Yaskawa INFORM job: R1_W72(-45,-90)KM-OK.JBI

/JOB
//NAME R1_W72(-45,-90)KM-OK
///FOLDERNAME KRIS-SCIANA
//POS
///NPOS 53,53,0,3,0,0
///TOOL 0
///POSTYPE PULSE
///PULSE
C00000=36093,-75117,-81688,-11832,61081,86345
C00001=121104,44356,-7752,-12211,112465,-19608
C00002=119726,72138,43556,-10749,114411,-20166
C00003=119728,72136,43553,-10749,114412,-20165
C00004=119725,70669,42344,-10765,114400,-20167
C00005=119722,69699,41648,-10758,114329,-20162
C00006=119729,72135,43552,-10749,114412,-20165
C00007=119732,73139,45374,238,113164,-19196
C00008=119737,74863,48427,239,112171,-19195
C00009=119729,72149,43570,239,113767,-19196
C00010=119729,72151,43571,239,113767,-19196
C00011=119726,72154,43576,238,113766,-19197
C00012=119720,72050,43451,519,96127,-46739
C00013=119722,72046,43446,519,96127,-46738
C00014=119749,73240,45977,517,95186,-46732
C00015=119747,72245,45197,517,95155,-46733
C00016=119749,73240,45977,517,95186,-46732
C00017=119752,74055,47327,517,94791,-46731
C00018=119723,72046,43446,519,96127,-46738
C00019=120494,78461,48464,494,96331,-46477
C00020=119130,74927,48027,540,94793,-46944
C00021=119532,76159,50009,527,94206,-46810
C00022=119725,72063,42900,520,96472,-46736
C00023=119723,72059,43462,519,96125,-46738
C00024=119720,72050,43451,519,96127,-46739
C00025=111817,-20677,-39808,24253,85188,64897
C00026=111822,-19931,-22646,24848,75884,62962
C00027=112411,-19087,-17904,24992,73443,62659
C00028=114208,-18286,-15193,24758,71757,62983
C00029=112577,-20422,-18113,25024,72884,62602
C00030=112592,-17414,-15899,24999,73047,62642
C00031=121850,-20195,-19127,22874,70872,65755
C00032=123019,-19624,-16008,35594,68743,65736
C00033=124000,-19465,-16017,35353,68407,66051
C00034=132626,-19286,-23113,19634,70806,69841
C00035=132624,-19877,-27646,19383,73156,70233
C00036=132617,-18981,-43608,18753,82905,71779
C00037=146857,37210,8702,-2862,82235,84576
C00038=151620,40537,21131,-4164,76490,86342
C00039=132754,24408,9297,18230,71766,81052
C00040=132688,21182,6297,18231,71962,81057
C00041=149891,38031,19022,-3707,76420,85748
C00042=144260,30621,12309,-2195,76538,83807
C00043=133734,23324,8789,17071,71503,81297
C00044=129277,26773,17464,28962,70643,78849
C00045=128722,27699,18908,29167,70475,78580
C00046=128434,28306,19806,29277,70363,78434
C00047=126520,32921,27495,30153,68979,77273
C00048=125069,31733,21247,29905,72303,77591
C00049=132931,22667,5718,20812,73042,80433
C00050=132926,24201,-9445,20133,82555,82064
C00051=133640,-149889,-134538,23781,27066,80448
C00052=14699,-137472,-132764,21891,29007,-82314
BC00000=211021,796909,1075051
BC00001=358765,1108219,959972
BC00002=358765,1108219,959972
BC00003=358096,1108178,933184
BC00004=357829,1108161,922465
BC00005=357829,1108161,922465
BC00006=357829,1108161,922468
BC00007=375276,1110547,921864
BC00008=375276,1110547,921864
BC00009=375276,1110547,921864
BC00010=376088,1110613,932260
BC00011=378119,1110780,958248
BC00012=250469,1133131,1039434
BC00013=247494,1133429,1014518
BC00014=246304,1133549,1004552
BC00015=246304,1133549,1004552
BC00016=246304,1133549,1004552
BC00017=246304,1133549,1004552
BC00018=248643,1134555,1002542
BC00019=263983,1135762,997435
BC00020=263980,1130615,977059
BC00021=263980,1130615,977059
BC00022=263980,1130615,977059
BC00023=263983,1135762,997435
BC00024=250469,1133131,1039434
BC00025=395849,1067691,1070910
BC00026=395849,1067691,1070910
BC00027=395849,1067587,1070910
BC00028=395849,1067544,1070905
BC00029=395849,1067545,1070910
BC00030=395849,1067545,1070910
BC00031=363979,1062628,1070905
BC00032=328518,1057159,1070910
BC00033=328518,1057159,1070910
BC00034=328755,1057154,1070910
BC00035=330110,1057258,1070910
BC00036=330110,1057258,1070910
BC00037=320330,1111284,1070909
BC00038=320328,1111285,1070910
BC00039=320328,1111285,1070910
BC00040=320328,1111285,1070910
BC00041=320328,1111285,1070910
BC00042=320328,1111285,1070910
BC00043=320328,1111285,1070910
BC00044=333958,1108190,1070910
BC00045=333958,1108190,1070910
BC00046=333958,1108190,1070910
BC00047=333958,1108190,1070910
BC00048=333967,1108189,1070910
BC00049=337587,1107891,1070910
BC00050=337587,1107891,1070910
BC00051=337586,1107893,1070908
BC00052=152981,671279,1070908
///POSTYPE BASE
///RECTAN
///RCONF 0,0,0,0,0,0,0,0,0,0,0,0,0,0,0,0,0,0,0,0,0,0,0,0
P00006=0.222,-3.123,-1.508,0.0000,0.0000,0.0000
P00021=-0.225,-6.128,-0.405,0.0000,0.0000,0.0000
P00022=0.222,-3.123,-1.508,0.0000,0.0000,0.0000
//INST
///DATE 2024/07/30 10:43
///ATTR SC,RW
///GROUP1 RB1,BS1
NOP
'r1_W72(-45,-90)
'Path S891
SFTOF
MOVJ C00000 BC00000 VJ=100.00
MOVJ C00001 BC00001 VJ=100.00
MOVJ C00002 BC00002 VJ=100.00
MOVJ C00003 BC00003 VJ=100.00
MOVL C00004 BC00004 V=60.0
REFP 3 C00005 BC00005
CALL JOB:SEARCH-R1
SET P022 P006
SFTON P022
MOVL C00006 BC00006 V=60.0
MOVL C00007 BC00007 V=60.0
REFP 3 C00008 BC00008
CALL JOB:SEARCH-R1
SET P022 P006
SFTON P022
MOVL C00009 BC00009 V=60.0
MOVL C00010 BC00010 V=166.7
MOVL C00011 BC00011 V=166.7
'Path S1463
SFTOF
MOVJ C00012 BC00012 VJ=100.00
MOVJ C00013 BC00013 VJ=100.00
MOVL C00014 BC00014 V=60.0
REFP 3 C00015 BC00015
CALL JOB:SEARCH-R1
SET P021 P006
SFTON P021
MOVL C00016 BC00016 V=50.0
REFP 3 C00017 BC00017
CALL JOB:SEARCH-R1
SET P021 P006
SFTON P021
MOVL C00018 BC00018 V=60.0
MOVL C00019 BC00019 V=100.0
MOVL C00020 BC00020 V=60.0
REFP 3 C00021 BC00021
CALL JOB:SEARCH-R1
SET P021 P006
SFTON P021
MOVL C00022 BC00022 V=60.0
MOVL C00023 BC00023 V=100.0
MOVL C00024 BC00024 V=1000.0
'Path W19
SFTOF
SFTON P022
MOVJ C00025 BC00025 VJ=100.00
MOVJ C00026 BC00026 VJ=100.00
MOVJ C00027 BC00027 VJ=100.00
MOVL C00028 BC00028 V=100.0 PL=0
REFP 1 C00029 BC00029
REFP 2 C00030 BC00030
MACRO1 MJ#(0) ARGF9
ARCON
SFTON P021
MOVL C00031 BC00031 V=10.8
MOVL C00032 BC00032 V=10.8
MOVL C00033 BC00033 V=10.8
ARCOF
MOVL C00034 BC00034 V=166.7
SFTOF
MOVL C00035 BC00035 V=166.7
MOVL C00036 BC00036 V=166.7
SFTON P021
MOVJ C00037 BC00037 VJ=50.00
MOVL C00038 BC00038 V=100.0 PL=0
REFP 1 C00039 BC00039
REFP 2 C00040 BC00040
MACRO1 MJ#(0) ARGF7
ARCON
MOVL C00041 BC00041 V=10.8
MOVL C00042 BC00042 V=10.8
MOVL C00043 BC00043 V=10.8
MOVL C00044 BC00044 V=10.8
MOVL C00045 BC00045 V=10.8
MOVL C00046 BC00046 V=10.8
MOVL C00047 BC00047 V=10.8
ARCOF
MOVL C00048 BC00048 V=166.7
MOVL C00049 BC00049 V=166.7
MOVL C00050 BC00050 V=166.7
SFTOF
MOVJ C00051 BC00051 VJ=100.00
MOVJ C00052 BC00052 VJ=100.00
END
